DATA_BLOCK "DiagnosticDataBlock"
VAR
  DP : STRUCT
    DPReadStatus : Int;
    Status : Array[0..1023] of Bool;
  END_STRUCT;
  Profinet : STRUCT
    PNReadStatus : Int;
    Status : Array[0..1023] of Bool;
  END_STRUCT;
END_VAR
BEGIN
END_DATA_BLOCK
